THIS^.testConvertVolume(
	sourceValue := 1.0,
	sourceUnit := CNM_RecipeHandling.VolumeUnit.LITER,
	sourcePrefix := CNM_RecipeHandling.MetricPrefixes.NONE,
	expectedValue := 1000.0,
	expectedUnit := CNM_RecipeHandling.VolumeUnit.LITER,
	expectedPrefix:= CNM_RecipeHandling.MetricPrefixes.MILLI
);
THIS^.testConvertVolume(
	sourceValue := 1.0,
	sourceUnit := CNM_RecipeHandling.VolumeUnit.LITER,
	sourcePrefix := CNM_RecipeHandling.MetricPrefixes.NONE,
	expectedValue := 0.001,
	expectedUnit := CNM_RecipeHandling.VolumeUnit.CUBIC_METER,
	expectedPrefix:= CNM_RecipeHandling.MetricPrefixes.NONE
);
THIS^.testConvertVolume(
	sourceValue := 1.0,
	sourceUnit := CNM_RecipeHandling.VolumeUnit.LITER,
	sourcePrefix := CNM_RecipeHandling.MetricPrefixes.NONE,
	expectedValue := 0.264172 ,
	expectedUnit := CNM_RecipeHandling.VolumeUnit.US_GALLON,
	expectedPrefix:= CNM_RecipeHandling.MetricPrefixes.NONE
);
THIS^.testConvertVolume(
	sourceValue := 1.0,
	sourceUnit := CNM_RecipeHandling.VolumeUnit.LITER,
	sourcePrefix := CNM_RecipeHandling.MetricPrefixes.NONE,
	expectedValue := 0.219969 ,
	expectedUnit := CNM_RecipeHandling.VolumeUnit.US_DRY_GALLON,
	expectedPrefix:= CNM_RecipeHandling.MetricPrefixes.NONE
);
THIS^.testConvertVolume(
	sourceValue := 1.0,
	sourceUnit := CNM_RecipeHandling.VolumeUnit.LITER,
	sourcePrefix := CNM_RecipeHandling.MetricPrefixes.NONE,
	expectedValue := 1.8161708314990030466 ,
	expectedUnit := CNM_RecipeHandling.VolumeUnit.US_DRY_PINT,
	expectedPrefix:= CNM_RecipeHandling.MetricPrefixes.NONE
);
THIS^.testConvertVolume(
	sourceValue := 1.0,
	sourceUnit := CNM_RecipeHandling.VolumeUnit.US_DRY_PINT,
	sourcePrefix := CNM_RecipeHandling.MetricPrefixes.NONE,
	expectedValue :=  1.16365 ,
	expectedUnit := CNM_RecipeHandling.VolumeUnit.US_PINT,
	expectedPrefix:= CNM_RecipeHandling.MetricPrefixes.NONE
);
THIS^.testConvertVolume(
	sourceValue := 1.0,
	sourceUnit := CNM_RecipeHandling.VolumeUnit.LITER,
	sourcePrefix := CNM_RecipeHandling.MetricPrefixes.NONE,
	expectedValue :=  0.00130795,
	expectedUnit := CNM_RecipeHandling.VolumeUnit.US_CUBIC_YARD,
	expectedPrefix:= CNM_RecipeHandling.MetricPrefixes.NONE
);
THIS^.testConvertVolume(
	sourceValue := 1.0,
	sourceUnit := CNM_RecipeHandling.VolumeUnit.LITER,
	sourcePrefix := CNM_RecipeHandling.MetricPrefixes.NONE,
	expectedValue :=  0.03531467,
	expectedUnit := CNM_RecipeHandling.VolumeUnit.US_CUBIC_FOOT,
	expectedPrefix:= CNM_RecipeHandling.MetricPrefixes.NONE
);
THIS^.testConvertVolume(
	sourceValue := 0.0,
	sourceUnit := CNM_RecipeHandling.VolumeUnit.LITER,
	sourcePrefix := CNM_RecipeHandling.MetricPrefixes.NONE,
	expectedValue :=  0.0,
	expectedUnit := CNM_RecipeHandling.VolumeUnit.LITER,
	expectedPrefix:= CNM_RecipeHandling.MetricPrefixes.MILLI
);
THIS^.testConvertVolume(
	sourceValue := 0.0,
	sourceUnit := CNM_RecipeHandling.VolumeUnit.LITER,
	sourcePrefix := CNM_RecipeHandling.MetricPrefixes.NONE,
	expectedValue :=  0.0,
	expectedUnit := CNM_RecipeHandling.VolumeUnit.US_GALLON,
	expectedPrefix:= CNM_RecipeHandling.MetricPrefixes.MILLI
);
THIS^.testConvertVolume(
	sourceValue := 0.0,
	sourceUnit := CNM_RecipeHandling.VolumeUnit.LITER,
	sourcePrefix := CNM_RecipeHandling.MetricPrefixes.NONE,
	expectedValue :=  0.0,
	expectedUnit := CNM_RecipeHandling.VolumeUnit.US_DRY_GALLON,
	expectedPrefix:= CNM_RecipeHandling.MetricPrefixes.MILLI
);
THIS^.testConvertVolume(
	sourceValue := 1000.0,
	sourceUnit := CNM_RecipeHandling.VolumeUnit.LITER,
	sourcePrefix := CNM_RecipeHandling.MetricPrefixes.NONE,
	expectedValue :=  1000000.0,
	expectedUnit := CNM_RecipeHandling.VolumeUnit.LITER,
	expectedPrefix:= CNM_RecipeHandling.MetricPrefixes.MILLI
);
THIS^.testConvertVolume(
	sourceValue := 1000.0,
	sourceUnit := CNM_RecipeHandling.VolumeUnit.LITER,
	sourcePrefix := CNM_RecipeHandling.MetricPrefixes.NONE,
	expectedValue :=  1.0,
	expectedUnit := CNM_RecipeHandling.VolumeUnit.CUBIC_METER,
	expectedPrefix:= CNM_RecipeHandling.MetricPrefixes.NONE
);
THIS^.testConvertVolume(
	sourceValue := 1000.0,
	sourceUnit := CNM_RecipeHandling.VolumeUnit.LITER,
	sourcePrefix := CNM_RecipeHandling.MetricPrefixes.NONE,
	expectedValue := 264.172,
	expectedUnit := CNM_RecipeHandling.VolumeUnit.US_GALLON,
	expectedPrefix:= CNM_RecipeHandling.MetricPrefixes.NONE
);
THIS^.testConvertVolume(
	sourceValue := 1000.0,
	sourceUnit := CNM_RecipeHandling.VolumeUnit.LITER,
	sourcePrefix := CNM_RecipeHandling.MetricPrefixes.NONE,
	expectedValue := 227.020746,
	expectedUnit := CNM_RecipeHandling.VolumeUnit.US_DRY_GALLON,
	expectedPrefix:= CNM_RecipeHandling.MetricPrefixes.NONE
);
THIS^.testConvertVolume(
	sourceValue := -1.0,
	sourceUnit := CNM_RecipeHandling.VolumeUnit.LITER,
	sourcePrefix := CNM_RecipeHandling.MetricPrefixes.NONE,
	expectedValue := -1000.0,
	expectedUnit := CNM_RecipeHandling.VolumeUnit.LITER,
	expectedPrefix:= CNM_RecipeHandling.MetricPrefixes.MILLI
);
THIS^.testConvertVolume(
	sourceValue := -1.0,
	sourceUnit := CNM_RecipeHandling.VolumeUnit.LITER,
	sourcePrefix := CNM_RecipeHandling.MetricPrefixes.NONE,
	expectedValue := -0.264172,
	expectedUnit := CNM_RecipeHandling.VolumeUnit.US_GALLON,
	expectedPrefix:= CNM_RecipeHandling.MetricPrefixes.NONE
);
THIS^.testConvertVolume(
	sourceValue := 1.0,
	sourceUnit := CNM_RecipeHandling.VolumeUnit.LITER,
	sourcePrefix := CNM_RecipeHandling.MetricPrefixes.KILO,
	expectedValue := 0.26417205,
	expectedUnit := CNM_RecipeHandling.VolumeUnit.US_GALLON,
	expectedPrefix:= CNM_RecipeHandling.MetricPrefixes.KILO
);
THIS^.testConvertVolume(
	sourceValue := 1.0,
	sourceUnit := CNM_RecipeHandling.VolumeUnit.CUBIC_METER,
	sourcePrefix := CNM_RecipeHandling.MetricPrefixes.NONE,
	expectedValue := 6.28981,
	expectedUnit := CNM_RecipeHandling.VolumeUnit.US_OIL_BARREL,
	expectedPrefix:= CNM_RecipeHandling.MetricPrefixes.NONE
);
THIS^.testConvertVolume(
	sourceValue := 1.0,
	sourceUnit := CNM_RecipeHandling.VolumeUnit.CUBIC_METER,
	sourcePrefix := CNM_RecipeHandling.MetricPrefixes.KILO,
	expectedValue := 6289810771.5398332750,
	expectedUnit := CNM_RecipeHandling.VolumeUnit.US_OIL_BARREL,
	expectedPrefix:= CNM_RecipeHandling.MetricPrefixes.NONE
);
THIS^.testConvertVolume(
	sourceValue := 3.14,
	sourceUnit := CNM_RecipeHandling.VolumeUnit.CUBIC_METER,
	sourcePrefix := CNM_RecipeHandling.MetricPrefixes.NONE,
	expectedValue := 19.75,
	expectedUnit := CNM_RecipeHandling.VolumeUnit.US_OIL_BARREL,
	expectedPrefix:= CNM_RecipeHandling.MetricPrefixes.NONE
);
THIS^.testConvertVolume(
	sourceValue := 1.41,
	sourceUnit := CNM_RecipeHandling.VolumeUnit.LITER,
	sourcePrefix := CNM_RecipeHandling.MetricPrefixes.NONE,
	expectedValue := 0.0088937924,
	expectedUnit := CNM_RecipeHandling.VolumeUnit.US_OIL_BARREL,
	expectedPrefix:= CNM_RecipeHandling.MetricPrefixes.NONE
);
THIS^.testConvertVolume(
	sourceValue := 1.0,
	sourceUnit := CNM_RecipeHandling.VolumeUnit.US_OIL_BARREL,
	sourcePrefix := CNM_RecipeHandling.MetricPrefixes.NONE,
	expectedValue := 0.1589872949,
	expectedUnit := CNM_RecipeHandling.VolumeUnit.CUBIC_METER,
	expectedPrefix:= CNM_RecipeHandling.MetricPrefixes.NONE
);
THIS^.testConvertVolume(
	sourceValue := 3.14,
	sourceUnit := CNM_RecipeHandling.VolumeUnit.US_OIL_BARREL,
	sourcePrefix := CNM_RecipeHandling.MetricPrefixes.NONE,
	expectedValue := 16880.6289,
	expectedUnit := CNM_RecipeHandling.VolumeUnit.US_FLUID_OUNCE,
	expectedPrefix:= CNM_RecipeHandling.MetricPrefixes.NONE
);
THIS^.testConvertVolume(
	sourceValue := THIS^.MINUS_ZERO,
	sourceUnit := CNM_RecipeHandling.VolumeUnit.LITER,
	sourcePrefix := CNM_RecipeHandling.MetricPrefixes.KILO,
	expectedValue := THIS^.MINUS_ZERO,
	expectedUnit := CNM_RecipeHandling.VolumeUnit.US_GALLON,
	expectedPrefix:= CNM_RecipeHandling.MetricPrefixes.KILO
);
THIS^.testConvertVolume(
	sourceValue := THIS^.MIN_SUBNORMAL,
	sourceUnit := CNM_RecipeHandling.VolumeUnit.LITER,
	sourcePrefix := CNM_RecipeHandling.MetricPrefixes.KILO,
	expectedValue := THIS^.MIN_SUBNORMAL,
	expectedUnit := CNM_RecipeHandling.VolumeUnit.US_GALLON,
	expectedPrefix:= CNM_RecipeHandling.MetricPrefixes.KILO
);
THIS^.testConvertVolume(
	sourceValue := THIS^.MAX_SUBNORMAL,
	sourceUnit := CNM_RecipeHandling.VolumeUnit.LITER,
	sourcePrefix := CNM_RecipeHandling.MetricPrefixes.KILO,
	expectedValue := THIS^.MAX_SUBNORMAL,
	expectedUnit := CNM_RecipeHandling.VolumeUnit.US_GALLON,
	expectedPrefix:= CNM_RecipeHandling.MetricPrefixes.KILO
);
THIS^.testConvertVolume(
	sourceValue := THIS^.SMALLEST_NEGATIVE_SUBNORMAL,
	sourceUnit := CNM_RecipeHandling.VolumeUnit.LITER,
	sourcePrefix := CNM_RecipeHandling.MetricPrefixes.KILO,
	expectedValue := THIS^.SMALLEST_NEGATIVE_SUBNORMAL,
	expectedUnit := CNM_RecipeHandling.VolumeUnit.US_GALLON,
	expectedPrefix:= CNM_RecipeHandling.MetricPrefixes.KILO
);
THIS^.testConvertVolume(
	sourceValue := THIS^.SMALLEST_POSITIVE_SUBNORMAL,
	sourceUnit := CNM_RecipeHandling.VolumeUnit.LITER,
	sourcePrefix := CNM_RecipeHandling.MetricPrefixes.KILO,
	expectedValue := THIS^.SMALLEST_POSITIVE_SUBNORMAL,
	expectedUnit := CNM_RecipeHandling.VolumeUnit.US_GALLON,
	expectedPrefix:= CNM_RecipeHandling.MetricPrefixes.KILO
);
THIS^.testConvertVolumeSpecialCases(
	sourceValue := THIS^.NAN,
	sourceUnit := CNM_RecipeHandling.VolumeUnit.LITER,
	sourcePrefix := CNM_RecipeHandling.MetricPrefixes.KILO,
	expectedValue := THIS^.NAN,
	expectedUnit := CNM_RecipeHandling.VolumeUnit.US_GALLON,
	expectedPrefix:= CNM_RecipeHandling.MetricPrefixes.KILO
);
THIS^.testConvertVolumeSpecialCases(
	sourceValue := THIS^.INF,
	sourceUnit := CNM_RecipeHandling.VolumeUnit.LITER,
	sourcePrefix := CNM_RecipeHandling.MetricPrefixes.KILO,
	expectedValue := THIS^.INF,
	expectedUnit := CNM_RecipeHandling.VolumeUnit.US_GALLON,
	expectedPrefix:= CNM_RecipeHandling.MetricPrefixes.KILO
);
THIS^.testConvertVolumeSpecialCases(
	sourceValue := THIS^.MINUS_INF,
	sourceUnit := CNM_RecipeHandling.VolumeUnit.LITER,
	sourcePrefix := CNM_RecipeHandling.MetricPrefixes.KILO,
	expectedValue := THIS^.MINUS_INF,
	expectedUnit := CNM_RecipeHandling.VolumeUnit.US_GALLON,
	expectedPrefix:= CNM_RecipeHandling.MetricPrefixes.KILO
);
TcUnit.TEST_FINISHED();
END_METHOD

(*

short summary
==================
This test method tests ``ConvertWeight``
method of CNM_RecipeHandling library with various inputs

.. <legal notes>

legal notes
=================
| SPDX-FileCopyrightText: © 2025 ekvip automation GmbH <info@ekvip.de>
| SPDX-License-Identifier: Apache-2.0
| For details check: Apache-2.0_

.. _Apache-2.0: https://www.apache.org/licenses/LICENSE-2.0

.. </legal notes>

*)

METHOD runConvertWeight
VAR_INPUT
END_VAR
RETURN(NOT TcUnit.TEST_ORDERED('testConvertWeight'));

THIS^.testConvertWeight(
	sourceWeightValue := 1.0,
	sourceWeightUnit := CNM_RecipeHandling.WeightUnit.GRAM,
	sourcePrefix := CNM_RecipeHandling.MetricPrefixes.NONE,
	expectedValue := 1.0,
	expectedUnit := CNM_RecipeHandling.WeightUnit.GRAM,
	expectedPrefix:= CNM_RecipeHandling.MetricPrefixes.NONE
);
THIS^.testConvertWeight(
	sourceWeightValue := 1.0,
	sourceWeightUnit := CNM_RecipeHandling.WeightUnit.GRAM,
	sourcePrefix := CNM_RecipeHandling.MetricPrefixes.KILO,
	expectedValue := 1000.0,
	expectedUnit := CNM_RecipeHandling.WeightUnit.GRAM,
	expectedPrefix:= CNM_RecipeHandling.MetricPrefixes.NONE
);
THIS^.testConvertWeight(
	sourceWeightValue := 1.0,
	sourceWeightUnit := CNM_RecipeHandling.WeightUnit.GRAM,
	sourcePrefix := CNM_RecipeHandling.MetricPrefixes.KILO,
	expectedValue := 1000.0,
	expectedUnit := CNM_RecipeHandling.WeightUnit.GRAM,
	expectedPrefix:= CNM_RecipeHandling.MetricPrefixes.NONE
);
THIS^.testConvertWeight(
	sourceWeightValue := 1.0,
	sourceWeightUnit := CNM_RecipeHandling.WeightUnit.GRAM,
	sourcePrefix := CNM_RecipeHandling.MetricPrefixes.KILO,
	expectedValue := 0.001,
	expectedUnit := CNM_RecipeHandling.WeightUnit.TON,
	expectedPrefix:= CNM_RecipeHandling.MetricPrefixes.NONE
);
THIS^.testConvertWeight(
	sourceWeightValue := 0.001,
	sourceWeightUnit := CNM_RecipeHandling.WeightUnit.TON,
	sourcePrefix := CNM_RecipeHandling.MetricPrefixes.NONE,
	expectedValue := 2.20462,
	expectedUnit := CNM_RecipeHandling.WeightUnit.US_POUND,
	expectedPrefix:= CNM_RecipeHandling.MetricPrefixes.NONE
);
THIS^.testConvertWeight(
	sourceWeightValue := 1.0,
	sourceWeightUnit := CNM_RecipeHandling.WeightUnit.GRAM,
	sourcePrefix := CNM_RecipeHandling.MetricPrefixes.KILO,
	expectedValue := 35.274,
	expectedUnit := CNM_RecipeHandling.WeightUnit.US_OUNCE,
	expectedPrefix:= CNM_RecipeHandling.MetricPrefixes.NONE
);
THIS^.testConvertWeight(
	sourceWeightValue := 1.0,
	sourceWeightUnit := CNM_RecipeHandling.WeightUnit.GRAM,
	sourcePrefix := CNM_RecipeHandling.MetricPrefixes.NONE,
	expectedValue := 1000,
	expectedUnit := CNM_RecipeHandling.WeightUnit.GRAM,
	expectedPrefix:= CNM_RecipeHandling.MetricPrefixes.MILLI
);
THIS^.testConvertWeight(
	sourceWeightValue := 1.0,
	sourceWeightUnit := CNM_RecipeHandling.WeightUnit.GRAM,
	sourcePrefix := CNM_RecipeHandling.MetricPrefixes.NONE,
	expectedValue := 0.00220462,
	expectedUnit := CNM_RecipeHandling.WeightUnit.US_POUND,
	expectedPrefix:= CNM_RecipeHandling.MetricPrefixes.NONE
);
THIS^.testConvertWeight(
	sourceWeightValue := 1.0,
	sourceWeightUnit := CNM_RecipeHandling.WeightUnit.GRAM,
	sourcePrefix := CNM_RecipeHandling.MetricPrefixes.NONE,
	expectedValue := 0.035274,
	expectedUnit := CNM_RecipeHandling.WeightUnit.US_OUNCE,
	expectedPrefix:= CNM_RecipeHandling.MetricPrefixes.NONE
);
THIS^.testConvertWeight(
	sourceWeightValue := 0.0,
	sourceWeightUnit := CNM_RecipeHandling.WeightUnit.GRAM,
	sourcePrefix := CNM_RecipeHandling.MetricPrefixes.KILO,
	expectedValue := 0.0,
	expectedUnit := CNM_RecipeHandling.WeightUnit.GRAM,
	expectedPrefix:= CNM_RecipeHandling.MetricPrefixes.NONE
);
THIS^.testConvertWeight(
	sourceWeightValue := 0.0,
	sourceWeightUnit := CNM_RecipeHandling.WeightUnit.GRAM,
	sourcePrefix := CNM_RecipeHandling.MetricPrefixes.KILO,
	expectedValue := 0.0,
	expectedUnit := CNM_RecipeHandling.WeightUnit.US_POUND,
	expectedPrefix:= CNM_RecipeHandling.MetricPrefixes.NONE
);
THIS^.testConvertWeight(
	sourceWeightValue := 1000.0,
	sourceWeightUnit := CNM_RecipeHandling.WeightUnit.GRAM,
	sourcePrefix := CNM_RecipeHandling.MetricPrefixes.KILO,
	expectedValue := 1.0,
	expectedUnit := CNM_RecipeHandling.WeightUnit.TON,
	expectedPrefix:= CNM_RecipeHandling.MetricPrefixes.NONE
);
THIS^.testConvertWeight(
	sourceWeightValue := 1000.0,
	sourceWeightUnit := CNM_RecipeHandling.WeightUnit.GRAM,
	sourcePrefix := CNM_RecipeHandling.MetricPrefixes.KILO,
	expectedValue := 2204.62,
	expectedUnit := CNM_RecipeHandling.WeightUnit.US_POUND,
	expectedPrefix:= CNM_RecipeHandling.MetricPrefixes.NONE
);
THIS^.testConvertWeight(
	sourceWeightValue := 1000.0,
	sourceWeightUnit := CNM_RecipeHandling.WeightUnit.GRAM,
	sourcePrefix := CNM_RecipeHandling.MetricPrefixes.KILO,
	expectedValue := 35273.96195,
	expectedUnit := CNM_RecipeHandling.WeightUnit.US_OUNCE,
	expectedPrefix:= CNM_RecipeHandling.MetricPrefixes.NONE
);
THIS^.testConvertWeight(
	sourceWeightValue := -1.0,
	sourceWeightUnit := CNM_RecipeHandling.WeightUnit.GRAM,
	sourcePrefix := CNM_RecipeHandling.MetricPrefixes.KILO,
	expectedValue := -1000,
	expectedUnit := CNM_RecipeHandling.WeightUnit.GRAM,
	expectedPrefix:= CNM_RecipeHandling.MetricPrefixes.NONE
);
THIS^.testConvertWeight(
	sourceWeightValue := -1.0,
	sourceWeightUnit := CNM_RecipeHandling.WeightUnit.GRAM,
	sourcePrefix := CNM_RecipeHandling.MetricPrefixes.KILO,
	expectedValue := -35.274,
	expectedUnit := CNM_RecipeHandling.WeightUnit.US_OUNCE,
	expectedPrefix:= CNM_RecipeHandling.MetricPrefixes.NONE
);
THIS^.testConvertWeight(
	sourceWeightValue := 1.0,
	sourceWeightUnit := CNM_RecipeHandling.WeightUnit.GRAM,
	sourcePrefix := CNM_RecipeHandling.MetricPrefixes.MEGA,
	expectedValue := 1000.0,
	expectedUnit := CNM_RecipeHandling.WeightUnit.GRAM,
	expectedPrefix:= CNM_RecipeHandling.MetricPrefixes.KILO
);
THIS^.testConvertWeight(
	sourceWeightValue := 1.0,
	sourceWeightUnit := CNM_RecipeHandling.WeightUnit.GRAM,
	sourcePrefix := CNM_RecipeHandling.MetricPrefixes.HECTO,
	expectedValue := 100.0,
	expectedUnit := CNM_RecipeHandling.WeightUnit.GRAM,
	expectedPrefix:= CNM_RecipeHandling.MetricPrefixes.NONE
);
THIS^.testConvertWeight(
	sourceWeightValue := 1.0,
	sourceWeightUnit := CNM_RecipeHandling.WeightUnit.GRAM,
	sourcePrefix := CNM_RecipeHandling.MetricPrefixes.DEKA,
	expectedValue := 10.0,
	expectedUnit := CNM_RecipeHandling.WeightUnit.GRAM,
	expectedPrefix:= CNM_RecipeHandling.MetricPrefixes.NONE
);
THIS^.testConvertWeight(
	sourceWeightValue := 1.0,
	sourceWeightUnit := CNM_RecipeHandling.WeightUnit.GRAM,
	sourcePrefix := CNM_RecipeHandling.MetricPrefixes.DECI,
	expectedValue := 0.1,
	expectedUnit := CNM_RecipeHandling.WeightUnit.GRAM,
	expectedPrefix:= CNM_RecipeHandling.MetricPrefixes.NONE
);
THIS^.testConvertWeight(
	sourceWeightValue := 1.0,
	sourceWeightUnit := CNM_RecipeHandling.WeightUnit.GRAM,
	sourcePrefix := CNM_RecipeHandling.MetricPrefixes.CENTI,
	expectedValue := 0.01,
	expectedUnit := CNM_RecipeHandling.WeightUnit.GRAM,
	expectedPrefix:= CNM_RecipeHandling.MetricPrefixes.NONE
);
THIS^.testConvertWeight(
	sourceWeightValue := 1.0,
	sourceWeightUnit := CNM_RecipeHandling.WeightUnit.GRAM,
	sourcePrefix := CNM_RecipeHandling.MetricPrefixes.KILO,
	expectedValue := 0.03527396,
	expectedUnit := CNM_RecipeHandling.WeightUnit.US_OUNCE,
	expectedPrefix:= CNM_RecipeHandling.MetricPrefixes.KILO
);
THIS^.testConvertWeight(
	sourceWeightValue := THIS^.MINUS_ZERO,
	sourceWeightUnit := CNM_RecipeHandling.WeightUnit.GRAM,
	sourcePrefix := CNM_RecipeHandling.MetricPrefixes.KILO,
	expectedValue := THIS^.MINUS_ZERO,
	expectedUnit := CNM_RecipeHandling.WeightUnit.GRAM,
	expectedPrefix:= CNM_RecipeHandling.MetricPrefixes.MILLI
);
THIS^.testConvertWeight(
	sourceWeightValue := THIS^.MIN_SUBNORMAL,
	sourceWeightUnit := CNM_RecipeHandling.WeightUnit.GRAM,
	sourcePrefix := CNM_RecipeHandling.MetricPrefixes.KILO,
	expectedValue := THIS^.MIN_SUBNORMAL,
	expectedUnit := CNM_RecipeHandling.WeightUnit.GRAM,
	expectedPrefix:= CNM_RecipeHandling.MetricPrefixes.MILLI
);
THIS^.testConvertWeight(
	sourceWeightValue := THIS^.MAX_SUBNORMAL,
	sourceWeightUnit := CNM_RecipeHandling.WeightUnit.GRAM,
	sourcePrefix := CNM_RecipeHandling.MetricPrefixes.KILO,
	expectedValue := THIS^.MAX_SUBNORMAL,
	expectedUnit := CNM_RecipeHandling.WeightUnit.GRAM,
	expectedPrefix:= CNM_RecipeHandling.MetricPrefixes.MILLI
);
THIS^.testConvertWeight(
	sourceWeightValue := THIS^.SMALLEST_NEGATIVE_SUBNORMAL,
	sourceWeightUnit := CNM_RecipeHandling.WeightUnit.GRAM,
	sourcePrefix := CNM_RecipeHandling.MetricPrefixes.KILO,
	expectedValue := THIS^.SMALLEST_NEGATIVE_SUBNORMAL,
	expectedUnit := CNM_RecipeHandling.WeightUnit.GRAM,
	expectedPrefix:= CNM_RecipeHandling.MetricPrefixes.MILLI
);
THIS^.testConvertWeight(
	sourceWeightValue := THIS^.SMALLEST_POSITIVE_SUBNORMAL,
	sourceWeightUnit := CNM_RecipeHandling.WeightUnit.GRAM,
	sourcePrefix := CNM_RecipeHandling.MetricPrefixes.KILO,
	expectedValue := THIS^.SMALLEST_POSITIVE_SUBNORMAL,
	expectedUnit := CNM_RecipeHandling.WeightUnit.GRAM,
	expectedPrefix:= CNM_RecipeHandling.MetricPrefixes.MILLI
);
THIS^.testConvertWightSpecialCases(
	sourceWeightValue := THIS^.NAN,
	sourceWeightUnit := CNM_RecipeHandling.WeightUnit.GRAM,
	sourcePrefix := CNM_RecipeHandling.MetricPrefixes.KILO,
	expectedValue := THIS^.NAN,
	expectedUnit := CNM_RecipeHandling.WeightUnit.GRAM,
	expectedPrefix:= CNM_RecipeHandling.MetricPrefixes.MILLI
);
THIS^.testConvertWightSpecialCases(
	sourceWeightValue := THIS^.INF,
	sourceWeightUnit := CNM_RecipeHandling.WeightUnit.GRAM,
	sourcePrefix := CNM_RecipeHandling.MetricPrefixes.KILO,
	expectedValue := THIS^.INF,
	expectedUnit := CNM_RecipeHandling.WeightUnit.GRAM,
	expectedPrefix:= CNM_RecipeHandling.MetricPrefixes.MILLI
);
THIS^.testConvertWightSpecialCases(
	sourceWeightValue := THIS^.MINUS_INF,
	sourceWeightUnit := CNM_RecipeHandling.WeightUnit.GRAM,
	sourcePrefix := CNM_RecipeHandling.MetricPrefixes.KILO,
	expectedValue := THIS^.MINUS_INF,
	expectedUnit := CNM_RecipeHandling.WeightUnit.GRAM,
	expectedPrefix:= CNM_RecipeHandling.MetricPrefixes.MILLI
);
TcUnit.TEST_FINISHED();
END_METHOD

(*

short summary
==================
This test method tests ``FastPow10``
method of CNM_RecipeHandling library with various inputs

.. <legal notes>

legal notes
=================
| SPDX-FileCopyrightText: © 2025 ekvip automation GmbH <info@ekvip.de>
| SPDX-License-Identifier: Apache-2.0
| For details check: Apache-2.0_

.. _Apache-2.0: https://www.apache.org/licenses/LICENSE-2.0

.. </legal notes>

*)

METHOD runFastPow10
VAR_INPUT
END_VAR
RETURN(NOT TcUnit.TEST_ORDERED('testFastPow10'));
THIS^.testFastPow10(
	exponentValue := 32,
	expectedFastPow10Value := 100000000000000000000000000000000.0
);
THIS^.testFastPow10(
	exponentValue := -5,
	expectedFastPow10Value := 0.00001
);
THIS^.testFastPow10(
	exponentValue := -3,
	expectedFastPow10Value := 0.001
);
THIS^.testFastPow10(
	exponentValue := -1, 
	expectedFastPow10Value := 0.1
);
THIS^.testFastPow10(
	exponentValue := 0,
	expectedFastPow10Value := 1.0
);
THIS^.testFastPow10(
	exponentValue := 1,
	expectedFastPow10Value := 10.0
);
THIS^.testFastPow10(
	exponentValue := 2, 
	expectedFastPow10Value := 100.0
);
THIS^.testFastPow10(
	exponentValue := 3, 
	expectedFastPow10Value := 1000.0
);
THIS^.testFastPow10(
	exponentValue := 6, 
	expectedFastPow10Value := 1000000.0
);
THIS^.testFastPow10(
	exponentValue := 9, 
	expectedFastPow10Value := 1000000000.0
);
THIS^.testFastPow10(
	exponentValue := 12, 
	expectedFastPow10Value := 1000000000000.0
);
THIS^.testFastPow10(
	exponentValue := -6, 
	expectedFastPow10Value := 0.000001
);
THIS^.testFastPow10(
	exponentValue := -9, 
	expectedFastPow10Value := 0.000000001
);
THIS^.testFastPow10(
	exponentValue := -12,
	expectedFastPow10Value := 0.000000000001
);
THIS^.testFastPow10(
	exponentValue := 15, 
	expectedFastPow10Value := 1000000000000000.0
);
THIS^.testFastPow10(
	exponentValue := -15, 
	expectedFastPow10Value := 0.000000000000001
);
THIS^.testFastPow10(
	exponentValue := 0,
	expectedFastPow10Value := 1.0
);
TcUnit.TEST_FINISHED();
END_METHOD

(*

short summary
==================
This test method tests ``CalculateVelocity``
method of CNM_RecipeHandling library, 
it provides the possibility to handover test data via parameter 


.. <legal notes>

legal notes
=================
| SPDX-FileCopyrightText: © 2025 ekvip automation GmbH <info@ekvip.de>
| SPDX-License-Identifier: Apache-2.0
| For details check: Apache-2.0_

.. _Apache-2.0: https://www.apache.org/licenses/LICENSE-2.0

.. </legal notes>

parameters
==========

*)
METHOD testCalculateVelocity
VAR_INPUT
	(* The distance traveled, in raw value (e.g. 100.0) *)
	distanceDeltaValue : LREAL;
	(* The time it took to travel the distance (e.g. 10.0 seconds) *)
	timeDeltaValue : LREAL ;
	(* Unit of distance (e.g. METER, MILE) *)
	distanceUnit : CNM_RecipeHandling.LengthUnit;
	(* Unit of time (e.g. SECONDS, MINUTES) *)
	timeUnit: CNM_RecipeHandling.DurationUnit;
	(* Metric prefix for distance (e.g. KILO for kilometers) *)
	distancePrefix : CNM_RecipeHandling.MetricPrefixes;
	(* Metric prefix for time (e.g. MILLI for milliseconds) *)
	timePrefix : CNM_RecipeHandling.MetricPrefixes;
	(* Expected result of velocity calculation (e.g. 10.0) *)
	expectedVelocityValue : LREAL;
	(* Expected distance unit in result (e.g. METER) *)
	expectedDistanceUnit :CNM_RecipeHandling.LengthUnit;
	(* Expected metric prefix for distance (e.g. NONE) *)
	expectedDistancePrefix : CNM_RecipeHandling.MetricPrefixes;
	(* Expected time unit in result (e.g. SECONDS) *)
	expectedDurationUnit:CNM_RecipeHandling.DurationUnit;
	(*  Expected prefix for duration (e.g. MILLI) *)
	expectedDurationPrefix : CNM_RecipeHandling.MetricPrefixes;
	(* just the expectation if the assertion to test must be worng or true *)
	//assertionShouldBeTrue :BOOL;
END_VAR
VAR
	sourceDistance : CNM_RecipeHandling.Length;
	sourceTime : CNM_RecipeHandling.Duration;
	libResult : CNM_RecipeHandling.Velocity;
END_VAR

sourceTime.unit := timeUnit;
sourceTime.prefix := timePrefix; 

sourceDistance.value := distanceDeltaValue;
sourceDistance.unit := distanceUnit;
sourceDistance.prefix := distancePrefix;

sourceTime.value := timeDeltaValue;
sourceTime.unit := timeUnit;
sourceTime.prefix := timePrefix;


libResult := CNM_RecipeHandling.CalculateVelocity(
	distanceDelta :=sourceDistance,
	timeDelta := sourceTime,
);

THIS^.AssertEquals_LREAL(
    Expected := expectedVelocityValue,
    Actual := libResult.value,
    Delta := 0.01,
   Message := SEL(expectedVelocityValue = libResult.value,
	CONCAT('CalculateVelocity value fail: exp velocity = ',CONCAT( TO_STRING(expectedVelocityValue), concat( ', act velocity value = ', TO_STRING(libResult.value))))
    ,'test is ok'));

THIS^.AssertEquals_INT(
	Expected := expectedDistancePrefix,
	Actual := libResult.distancePrefix,
    Message := SEL(expectedDistancePrefix = libResult.distancePrefix,
	CONCAT('CalculateVelocity prefix fail: exp distance prefix  = ',CONCAT( TO_STRING(expectedDistancePrefix), concat( ', act distance prefix = ', TO_STRING(libResult.distancePrefix))))
    ,'test is ok')
);

THIS^.AssertEquals_INT(
	Expected := expectedDistanceUnit,
	Actual := libResult.distanceUnit,
    Message := SEL(expectedDistanceUnit = libResult.distanceUnit,
	CONCAT('CalculateVelocity unit fail: exp distance unit = ',CONCAT( TO_STRING(expectedDistanceUnit), concat( ', act distance unit = ', TO_STRING(libResult.distanceUnit))))
    ,'test is ok')
);

THIS^.AssertEquals_INT(
	Expected := expectedDurationPrefix,
	Actual := libResult.timePrefix,
    Message := SEL(expectedDurationPrefix = libResult.timePrefix,
	CONCAT('CalculateVelocity prefix fail: exp duration Prefix = ',CONCAT( TO_STRING(expectedDurationPrefix), concat( ', act duration Prefix = ', TO_STRING(libResult.timePrefix))))
    ,'test is ok')
);

THIS^.AssertEquals_INT(
	Expected := expectedDurationUnit,
	Actual := libResult.timeUnit,
    Message := SEL(expectedDurationUnit = libResult.timeUnit,
	CONCAT('CalculateVelocity unit fail: exp duration Unit = ',CONCAT( TO_STRING(expectedDurationUnit), concat( ', act duration Unit = ', TO_STRING(libResult.timeUnit))))
    ,'test is ok')
);
END_METHOD

(*

short summary
==================
This test method tests ``CalculateVelocity``
method of CNM_RecipeHandling library for special cases, 
it provides the possibility to handover test data via parameter 


.. <legal notes>

legal notes
=================
| SPDX-FileCopyrightText: © 2025 ekvip automation GmbH <info@ekvip.de>
| SPDX-License-Identifier: Apache-2.0
| For details check: Apache-2.0_

.. _Apache-2.0: https://www.apache.org/licenses/LICENSE-2.0

.. </legal notes>

parameters
==========

*)

METHOD testCalculateVelocitySpecialCases
	VAR_INPUT
	(* The distance traveled, in raw value (e.g. 100.0) *)
	distanceDeltaValue : LREAL;
	(* The time it took to travel the distance (e.g. 10.0 seconds) *)
	timeDeltaValue : LREAL ;
	(* Unit of distance (e.g. METER, MILE) *)
	distanceUnit : CNM_RecipeHandling.LengthUnit;
	(* Unit of time (e.g. SECONDS, MINUTES) *)
	timeUnit: CNM_RecipeHandling.DurationUnit;
	(* Metric prefix for distance (e.g. KILO for kilometers) *)
	distancePrefix : CNM_RecipeHandling.MetricPrefixes;
	(* Metric prefix for time (e.g. MILLI for milliseconds) *)
	timePrefix : CNM_RecipeHandling.MetricPrefixes;
	(* Expected result of velocity calculation (e.g. 10.0) *)
	expectedVelocityValue : LREAL;
	(* Expected distance unit in result (e.g. METER) *)
	expectedDistanceUnit :CNM_RecipeHandling.LengthUnit;
	(* Expected metric prefix for distance (e.g. NONE) *)
	expectedDistancePrefix : CNM_RecipeHandling.MetricPrefixes;
	(* Expected time unit in result (e.g. SECONDS) *)
	expectedDurationUnit:CNM_RecipeHandling.DurationUnit;
	(*  Expected prefix for duration (e.g. MILLI) *)
	expectedDurationPrefix : CNM_RecipeHandling.MetricPrefixes;;
END_VAR
VAR
	sourceDistance : CNM_RecipeHandling.Length;
	sourceTime : CNM_RecipeHandling.Duration;
	libResult : CNM_RecipeHandling.Velocity;
	(* contains the format string for the test message *)
	//message :Tc2_System.T_MaxString := 'Test failed';
	//Actual: INT;
END_VAR
sourceTime.unit := timeUnit;
sourceTime.prefix := timePrefix; 

sourceDistance.value := distanceDeltaValue;
sourceDistance.unit := distanceUnit;
sourceDistance.prefix := distancePrefix;

sourceTime.value := timeDeltaValue;
sourceTime.unit := timeUnit;
sourceTime.prefix := timePrefix;

libResult := CNM_RecipeHandling.CalculateVelocity(
	distanceDelta :=sourceDistance,
	timeDelta := sourceTime,
);

IF Tc2_Utilities.LrealIsNaN(expectedVelocityValue) THEN
	AssertTrue(Condition := Tc2_Utilities.LrealIsNaN(libResult.value),
    Message := 'test faild assertion NaN should be true');
ELSIF NOT (Tc2_Utilities.LrealIsFinite(expectedVelocityValue))THEN
	 AssertTrue(Condition := NOT(Tc2_Utilities.LrealIsFinite(libResult.value)),
    Message := 'test faild assertion INF should be True');
END_IF
END_METHOD

METHOD testConvertAngle
VAR_INPUT
	(* The input value to convert (e.g. 3.14159) *)
	sourceValue : LREAL;
	(* The unit of the input angle (e.g. RADIANS, DEGREES) *)
	sourceUnit : CNM_RecipeHandling.AngleUnit;
	(* The expected result after conversion *)
	expectedValue : LREAL;
	(* The expected output unit *)
	expectedUnit :CNM_RecipeHandling.AngleUnit;
END_VAR
VAR
	sourceAngle : CNM_RecipeHandling.Angle;
	libResult : CNM_RecipeHandling.Angle;
	delta : LREAL;
END_VAR
// Setup test input
sourceAngle.value := sourceValue;
sourceAngle.unit := sourceUnit;

// Call the function to test
libResult := CNM_RecipeHandling.ConvertAngle(
	angleToConvert := sourceAngle,
	convertTo := expectedUnit
);

// Calculate appropriate delta based on magnitude of expected value
IF ABS(expectedValue) > 1000.0 THEN
	delta := 0.1; // Larger tolerance for large numbers (arc seconds)
ELSIF ABS(expectedValue) > 100.0 THEN
	delta := 0.01; // Medium tolerance for medium numbers
ELSIF ABS(expectedValue) > 1.0 THEN
	delta := 0.0001; // Small tolerance for normal numbers
ELSE
	delta := 0.000001; // Very small tolerance for small numbers
END_IF

// Verify the unit is correct
THIS^.AssertEquals_INT(
	Expected := expectedUnit,
	Actual := libResult.unit,
	Message := CONCAT('Unit conversion failed: expected ', 
		CONCAT(TO_STRING(expectedUnit), 
		CONCAT(', got ', TO_STRING(libResult.unit))))
);

// Verify the value is correct
THIS^.AssertEquals_LREAL(
	Expected := expectedValue,
	Actual := libResult.value,
	Delta := delta,
	Message := CONCAT('Value conversion failed: from ', 
		CONCAT(TO_STRING(sourceUnit), 
		CONCAT(', to ', TO_STRING(expectedUnit))))
);
END_METHOD

METHOD testConvertAngleSpecialCases
VAR_INPUT
	(* The input value to convert (e.g. NaN, Inf) *)
	sourceValue : LREAL;
	(* The unit of the input angle *)
	sourceUnit : CNM_RecipeHandling.AngleUnit;
	(* The expected result after conversion *)
	expectedValue : LREAL;
	(* The expected output unit *)
	expectedUnit :CNM_RecipeHandling.AngleUnit;
END_VAR
VAR
	sourceAngle : CNM_RecipeHandling.Angle;
	libResult : CNM_RecipeHandling.Angle;
END_VAR
// Setup test input
sourceAngle.value := sourceValue;
sourceAngle.unit := sourceUnit;

// Call the function to test
libResult := CNM_RecipeHandling.ConvertAngle(
	angleToConvert := sourceAngle,
	convertTo := expectedUnit
);

IF Tc2_Utilities.LrealIsNaN(expectedValue) THEN
	AssertTrue(Condition := Tc2_Utilities.LrealIsNaN(libResult.value),
    Message := 'test failed assertion NaN should be true');
ELSIF NOT (Tc2_Utilities.LrealIsFinite(expectedValue))THEN
	 AssertTrue(Condition := NOT(Tc2_Utilities.LrealIsFinite(libResult.value)),
    Message := 'test faild assertion INF should be True');
END_IF
END_METHOD

(*

short summary
==================
This test method tests ``ConvertAngularVelocity``
method of CNM_RecipeHandling library, 
it provides the possibility to handover test data via parameter 


.. <legal notes>

legal notes
=================
| SPDX-FileCopyrightText: © 2025 ekvip automation GmbH <info@ekvip.de>
| SPDX-License-Identifier: Apache-2.0
| For details check: Apache-2.0_

.. _Apache-2.0: https://www.apache.org/licenses/LICENSE-2.0

.. </legal notes>

parameters
==========

*)

METHOD testConvertAngularVelocity
VAR_INPUT
    (* Input velocity value to be converted, e.g. 10.0 *)
    sourceVelocityValue : LREAL; 
    (* Expected result after conversion, used for assertion *)
    expectedVelocityValue : LREAL;
    (* Unit of distance used in velocity, e.g. METER *)
    sourceUnit : CNM_RecipeHandling.AngleUnit;
    (* Expected unit of distance after conversion *)
    expectedAngleUnit : CNM_RecipeHandling.AngleUnit;
    (* Unit of time used in velocity, e.g. SECONDS *)
    sourceDurationUnit : CNM_RecipeHandling.DurationUnit;
    (* Metric prefix of the time input, e.g. MILLI *)
    sourceDurationPrefix : CNM_RecipeHandling.MetricPrefixes;
    (* Expected time unit after conversion *)
    expectedDurationUnit : CNM_RecipeHandling.DurationUnit;
    (* Expected time prefix after conversion *)
    expectedDurationPrefix : CNM_RecipeHandling.MetricPrefixes;
END_VAR
VAR
	sourceVelocity : CNM_RecipeHandling.AngularVelocity;
	libResult : CNM_RecipeHandling.AngularVelocity;
	sourcePrefix: CNM_RecipeHandling.MetricPrefixes;
END_VAR

//test-input
sourceVelocity.value := sourceVelocityValue;
sourceVelocity.angularDistanceUnit := sourceUnit;
sourceVelocity.timeUnit := sourceDurationUnit;
sourceVelocity.timePrefix := sourceDurationPrefix; 

//function to call
libResult := CNM_RecipeHandling.ConvertAngularVelocity(
	angularVelocityToConvert := sourceVelocity,
	convertAngleTo := expectedAngleUnit,
	convertTimeTo := expectedDurationUnit,
	resultPrefixTime := expectedDurationPrefix
);

THIS^.AssertEquals_LREAL(
    Expected := expectedVelocityValue,
    Actual := libResult.value,
    Delta := 0.01,
   Message := SEL(expectedVelocityValue = libResult.value,
	CONCAT('value fail: exp velocity value = ',CONCAT( TO_STRING(expectedVelocityValue), concat( ', act  velocity value = ', TO_STRING(libResult.value))))
    ,'test is ok'));

THIS^.AssertEquals_INT(
	Expected := expectedAngleUnit,
	Actual := libResult.angularDistanceUnit,
    Message := CONCAT('ConvertVelocity unit fail: exp distance unit = ',CONCAT( TO_STRING(expectedAngleUnit), concat( ', act distance unit = ', TO_STRING(libResult.angularDistanceUnit))))
);

THIS^.AssertEquals_INT(
	Expected := expectedDurationPrefix,
	Actual := libResult.timePrefix,
    Message := SEL(expectedDurationPrefix = libResult.timePrefix,
	CONCAT('ConvertVelocity prefix fail: exp duration Prefix = ',CONCAT( TO_STRING(expectedDurationPrefix), concat( ', act duration Prefix = ', TO_STRING(libResult.timePrefix))))
    ,'test is ok')
);
THIS^.AssertEquals_INT(
	Expected := expectedDurationUnit,
	Actual := libResult.timeUnit,
    Message := SEL(expectedDurationUnit = libResult.timeUnit,
	CONCAT('ConvertVelocity unit fail: exp duration Unit = ',CONCAT( TO_STRING(expectedDurationUnit), concat( ', act duration Unit = ', TO_STRING(libResult.timeUnit))))
    ,'test is ok')
);
END_METHOD

(*

short summary
==================
This test method tests ``ConvertVelocity``
method of CNM_RecipeHandling library for special cases, 
it provides the possibility to handover test data via parameter 


.. <legal notes>

legal notes
=================
| SPDX-FileCopyrightText: © 2025 ekvip automation GmbH <info@ekvip.de>
| SPDX-License-Identifier: Apache-2.0
| For details check: Apache-2.0_

.. _Apache-2.0: https://www.apache.org/licenses/LICENSE-2.0

.. </legal notes>

parameters
==========

*)

METHOD testConvertAngularVelocitySpecialCases
VAR_INPUT
    (* Input velocity value to be converted, e.g. 10.0 *)
    sourceVelocityValue : LREAL; 
    (* Expected result after conversion, used for assertion *)
    expectedVelocityValue : LREAL;
    (* Unit of distance used in velocity, e.g. METER *)
    sourceUnit : CNM_RecipeHandling.AngleUnit;
    (* Expected unit of distance after conversion *)
    expectedAngleUnit : CNM_RecipeHandling.AngleUnit;
    (* Unit of time used in velocity, e.g. SECONDS *)
    sourceDurationUnit : CNM_RecipeHandling.DurationUnit;
    (* Metric prefix of the time input, e.g. MILLI *)
    sourceDurationPrefix : CNM_RecipeHandling.MetricPrefixes;
    (* Expected time unit after conversion *)
    expectedDurationUnit : CNM_RecipeHandling.DurationUnit;
    (* Expected time prefix after conversion *)
    expectedDurationPrefix : CNM_RecipeHandling.MetricPrefixes;
END_VAR
VAR
	sourceVelocity : CNM_RecipeHandling.AngularVelocity;
	libResult : CNM_RecipeHandling.AngularVelocity;
	sourcePrefix: CNM_RecipeHandling.MetricPrefixes;
END_VAR
//test-input
sourceVelocity.value := sourceVelocityValue;
sourceVelocity.angularDistanceUnit := sourceUnit;
sourceVelocity.timeUnit := sourceDurationUnit;
sourceVelocity.timePrefix := sourceDurationPrefix; 

//function to call
libResult := CNM_RecipeHandling.ConvertAngularVelocity(
	angularVelocityToConvert:=sourceVelocity,
	convertAngleTo :=expectedAngleUnit,
	convertTimeTo := expectedDurationUnit,
	resultPrefixTime := expectedDurationPrefix
);

IF Tc2_Utilities.LrealIsNaN(expectedVelocityValue) THEN
	AssertTrue(Condition := Tc2_Utilities.LrealIsNaN(libResult.value),
    Message := 'test faild assertion NaN should be true');
ELSIF NOT (Tc2_Utilities.LrealIsFinite(expectedVelocityValue))THEN
	 AssertFalse(Condition := Tc2_Utilities.LrealIsFinite(libResult.value),
    Message := 'test faild assertion INF should be True');
END_IF
END_METHOD

(*

short summary
==================
This test method tests ``ConvertArea``
method of CNM_RecipeHandling library, 
it provides the possibility to handover test data via parameter 


.. <legal notes>

legal notes
=================
| SPDX-FileCopyrightText: © 2025 ekvip automation GmbH <info@ekvip.de>
| SPDX-License-Identifier: Apache-2.0
| For details check: Apache-2.0_

.. _Apache-2.0: https://www.apache.org/licenses/LICENSE-2.0

.. </legal notes>

parameters
==========

*)

METHOD testConvertArea
VAR_INPUT
	(* Input area value to be converted (e.g., 1.0) *)
	sourceValue : LREAL;
	(* Unit of the source area (e.g., SQUARE_METER, US_ACRE) *)
	sourceUnit : CNM_RecipeHandling.AreaUnit;
	(* Metric prefix of the source area unit (e.g., NONE, KILO, MILLI) *)
	sourcePrefix : CNM_RecipeHandling.MetricPrefixes;
	(* Expected result value after conversion *)
	expectedValue : LREAL;
	(* Target unit to which the area should be converted *)
	expectedUnit :CNM_RecipeHandling.AreaUnit;
	(* Metric prefix for the expected unit (e.g., NONE, MILLI) *)
	expectedPrefix : CNM_RecipeHandling.MetricPrefixes;
END_VAR
VAR
	sourceArea : CNM_RecipeHandling.Area;
	libResult : CNM_RecipeHandling.Area;
END_VAR
sourceArea.value := sourceValue;
sourceArea.unit := sourceUnit;
sourceArea.prefix := sourcePrefix;

libResult := CNM_RecipeHandling.ConvertArea(
	areaToconvert := sourceArea,
	convertTo := expectedUnit,
	resultPrefix := expectedPrefix
);

THIS^.AssertEquals_LREAL(
	Expected := expectedValue,
	Actual := libResult.value,
	Delta := 0.01,
   Message := SEL(expectedValue = libResult.value,
	CONCAT('normal case testConvertArea value fail: exp = ',CONCAT( TO_STRING(expectedValue), concat( ', act = ', TO_STRING(libResult.value))))
    ,'test is ok'))
;
THIS^.AssertEquals_INT(
	Expected := expectedPrefix,
	Actual := libResult.prefix,
    Message := SEL(expectedPrefix = libResult.prefix,
	CONCAT('normal case testConvertAre prefix fail: exp = ',CONCAT( TO_STRING(expectedPrefix), concat( ', act = ', TO_STRING(libResult.prefix))))
    ,'test is ok')
);

THIS^.AssertEquals_INT(
	Expected := expectedUnit,
	Actual := libResult.unit,
    Message := SEL(expectedUnit = libResult.unit,
	CONCAT('normal case testConvertAre unit fail: exp = ',CONCAT( TO_STRING(expectedUnit), concat( ', act = ', TO_STRING(libResult.unit))))
    ,'test is ok')
);
END_METHOD

(*

short summary
==================
This test method tests ``ConvertArea``
method of CNM_RecipeHandling library, 
it provides the possibility to handover test data via parameter 


.. <legal notes>

legal notes
=================
| SPDX-FileCopyrightText: © 2025 ekvip automation GmbH <info@ekvip.de>
| SPDX-License-Identifier: Apache-2.0
| For details check: Apache-2.0_

.. _Apache-2.0: https://www.apache.org/licenses/LICENSE-2.0

.. </legal notes>

parameters
==========

*)
METHOD testConvertAreaSpecialCases
VAR_INPUT
	(* Input area value to be converted (e.g., 1.0) *)
	sourceValue : LREAL;
	(* Unit of the source area (e.g., SQUARE_METER, US_ACRE) *)
	sourceUnit : CNM_RecipeHandling.AreaUnit;
	(* Metric prefix of the source area unit (e.g., NONE, KILO, MILLI) *)
	sourcePrefix : CNM_RecipeHandling.MetricPrefixes;
	(* Expected result value after conversion *)
	expectedValue : LREAL;
	(* Target unit to which the area should be converted *)
	expectedUnit :CNM_RecipeHandling.AreaUnit;
	(* Metric prefix for the expected unit (e.g., NONE, MILLI) *)
	expectedPrefix : CNM_RecipeHandling.MetricPrefixes;
END_VAR
VAR
	a :BOOL;
	input : CNM_RecipeHandling.Area;
	libResult : CNM_RecipeHandling.Area;
END_VAR
input.value := sourceValue;
input.unit := sourceUnit;
input.prefix := sourcePrefix;

libResult := CNM_RecipeHandling.ConvertArea(
	areaToconvert := input,
	convertTo := expectedUnit,
	resultPrefix := expectedPrefix
);

IF Tc2_Utilities.LrealIsNaN(expectedValue) THEN
	AssertTrue(Condition := Tc2_Utilities.LrealIsNaN(libResult.value),
    Message := 'test faild assertion NaN should be true');
ELSIF NOT (Tc2_Utilities.LrealIsFinite(expectedValue))THEN
	 AssertTrue(Condition := NOT(Tc2_Utilities.LrealIsFinite(libResult.value)),
    Message := 'test faild assertion INF should be True');
END_IF
END_METHOD

(*

short summary
==================
This test method tests ``ConvertDuration``
method of CNM_RecipeHandling library, 
it provides the possibility to handover test data via parameter 


.. <legal notes>

legal notes
=================
| SPDX-FileCopyrightText: © 2025 ekvip automation GmbH <info@ekvip.de>
| SPDX-License-Identifier: Apache-2.0
| For details check: Apache-2.0_

.. _Apache-2.0: https://www.apache.org/licenses/LICENSE-2.0

.. </legal notes>

parameters
==========

*)

METHOD testConvertDuration
VAR_INPUT
	(* The original time value to convert (e.g. 120.0) *)
	sourceValue : LREAL;
	(* The unit of the input time (e.g. SECONDS, MINUTES) *)
	sourceUnit : CNM_RecipeHandling.DurationUnit;
	(* The metric prefix for input time (e.g. MILLI for milliseconds) *)
	sourcePrefix : CNM_RecipeHandling.MetricPrefixes;
	(* The expected result value after conversion (e.g. 2.0) *)
	expectedValue : LREAL;
	(* The expected time unit after conversion (e.g. MINUTES) *)
	expectedUnit :CNM_RecipeHandling.DurationUnit;
	(* The expected metric prefix for the result (e.g. NONE) *)
	expectedPrefix : CNM_RecipeHandling.MetricPrefixes;
END_VAR
VAR
	sourceDuration : CNM_RecipeHandling.Duration;
	libResult : CNM_RecipeHandling.Duration;
END_VAR
sourceDuration.value := sourceValue;
sourceDuration.unit := sourceUnit;
sourceDuration.prefix := sourcePrefix;

libResult := CNM_RecipeHandling.ConvertDuration(
	durationToConvert :=sourceDuration,
	convertTo := expectedUnit,
	resultPrefix := expectedPrefix
);

THIS^.AssertEquals_LREAL(
    Expected := expectedValue,
    Actual := libResult.value,
    Delta := 0.01,
   Message := SEL(expectedValue = libResult.value,
	CONCAT('ConvertDuration value fail: exp = ',CONCAT( TO_STRING(expectedValue), concat( ', act = ', TO_STRING(libResult.value))))
    ,'test is ok'));

THIS^.AssertEquals_INT(
	Expected := expectedPrefix,
	Actual := libResult.prefix,
    Message := SEL(expectedPrefix = libResult.prefix,
	CONCAT('ConvertDuration prefix fail: exp = ',CONCAT( TO_STRING(expectedPrefix), concat( ', act = ', TO_STRING(libResult.prefix))))
    ,'test is ok')
);

THIS^.AssertEquals_INT(
	Expected := expectedUnit,
	Actual := libResult.unit,
    Message := SEL(expectedUnit = libResult.unit,
	CONCAT('ConvertDuration unit fail: exp = ',CONCAT( TO_STRING(expectedUnit), concat( ', act = ', TO_STRING(libResult.unit))))
    ,'test is ok')
);
END_METHOD

(*

short summary
==================
This test method tests ``ConvertDuration``
method of CNM_RecipeHandling library for special cases, 
it provides the possibility to handover test data via parameter 


.. <legal notes>

legal notes
=================
| SPDX-FileCopyrightText: © 2025 ekvip automation GmbH <info@ekvip.de>
| SPDX-License-Identifier: Apache-2.0
| For details check: Apache-2.0_

.. _Apache-2.0: https://www.apache.org/licenses/LICENSE-2.0

.. </legal notes>

parameters
==========

*)

METHOD testConvertDurationSpecialCases
VAR_INPUT
	(* The original time value to convert (e.g. 120.0) *)
	sourceValue : LREAL;
	(* The unit of the input time (e.g. SECONDS, MINUTES) *)
	sourceUnit : CNM_RecipeHandling.DurationUnit;
	(* The metric prefix for input time (e.g. MILLI for milliseconds) *)
	sourcePrefix : CNM_RecipeHandling.MetricPrefixes;
	(* The expected result value after conversion (e.g. 2.0) *)
	expectedValue : LREAL;
	(* The expected time unit after conversion (e.g. MINUTES) *)
	expectedUnit :CNM_RecipeHandling.DurationUnit;
	(* The expected metric prefix for the result (e.g. NONE) *)
	expectedPrefix : CNM_RecipeHandling.MetricPrefixes;
END_VAR
VAR
	sourceDuration : CNM_RecipeHandling.Duration;
	libResult : CNM_RecipeHandling.Duration;
END_VAR
sourceDuration.value := sourceValue;
sourceDuration.unit := sourceUnit;
sourceDuration.prefix := sourcePrefix;

libResult := CNM_RecipeHandling.ConvertDuration(
	durationToConvert :=sourceDuration,
	convertTo := expectedUnit,
	resultPrefix := expectedPrefix
);

IF Tc2_Utilities.LrealIsNaN(expectedValue) THEN
	AssertTrue(Condition := Tc2_Utilities.LrealIsNaN(libResult.value),
    Message := 'test faild assertion NaN should be true');
ELSIF NOT (Tc2_Utilities.LrealIsFinite(expectedValue))THEN
	 AssertTrue(Condition := NOT(Tc2_Utilities.LrealIsFinite(libResult.value)),
    Message := 'test faild assertion INF should be True');
END_IF
END_METHOD

(*

short summary
==================
This test method tests ``ConvertLength``
method of CNM_RecipeHandling library, 
it provides the possibility to handover test data via parameter 


.. <legal notes>

legal notes
=================
| SPDX-FileCopyrightText: © 2025 ekvip automation GmbH <info@ekvip.de>
| SPDX-License-Identifier: Apache-2.0
| For details check: Apache-2.0_

.. _Apache-2.0: https://www.apache.org/licenses/LICENSE-2.0

.. </legal notes>

parameters
==========

*)

METHOD testConvertLength
VAR_INPUT
	(* The input value to convert (e.g. 1.0) *)
	sourceValue : LREAL;
	(* The unit of the input length (e.g. METER, INCH) *)
	sourceUnit : CNM_RecipeHandling.LengthUnit;
	(* Metric prefix for the input value (e.g. MILLI, KILO) *)
	sourcePrefix : CNM_RecipeHandling.MetricPrefixes;
	(* The expected result after conversion (e.g. 1000.0) *)
	expectedValue : LREAL;
	(* The expected output unit (e.g. MILLIMETER) *)
	expectedUnit :CNM_RecipeHandling.LengthUnit;
	(* The expected metric prefix for the output (e.g. NONE) *)
	expectedPrefix : CNM_RecipeHandling.MetricPrefixes;
END_VAR
VAR
	sourceDistance : CNM_RecipeHandling.Length;
	libResult : CNM_RecipeHandling.Length;
END_VAR

//teat-input
sourceDistance.value := sourceValue;
sourceDistance.unit := sourceUnit;
sourceDistance.prefix := sourcePrefix;

//function to call
libResult := CNM_RecipeHandling.ConvertLength(
	lengthToConvert :=sourceDistance,
	convertTo := expectedUnit,
	resultPrefix := expectedPrefix
);

THIS^.AssertEquals_LREAL(
    Expected := expectedValue,
    Actual := libResult.value,
    Delta := 0.01,
   Message := SEL(expectedValue = libResult.value,
	CONCAT('ConvertLength value fail: exp = ',CONCAT( TO_STRING(expectedValue), concat( ', act = ', TO_STRING(libResult.value))))
    ,'test is ok'));


THIS^.AssertEquals_INT(
	Expected := expectedPrefix,
	Actual := libResult.prefix,
    Message := SEL(expectedPrefix = libResult.prefix,
	CONCAT('ConvertLength prefix fail: exp = ',CONCAT( TO_STRING(expectedPrefix), concat( ', act = ', TO_STRING(libResult.prefix))))
    ,'test is ok')
);
THIS^.AssertEquals_INT(
	Expected := expectedUnit,
	Actual := libResult.unit,
    Message := SEL(expectedUnit = libResult.unit,
	CONCAT('ConvertLength unit fail: exp = ',CONCAT( TO_STRING(expectedUnit), concat( ', act = ', TO_STRING(libResult.unit))))
    ,'test is ok')
);
END_METHOD

(*

short summary
==================
This test method tests ``ConvertLength``
method of CNM_RecipeHandling library for special cases, 
it provides the possibility to handover test data via parameter 


.. <legal notes>

legal notes
=================
| SPDX-FileCopyrightText: © 2025 ekvip automation GmbH <info@ekvip.de>
| SPDX-License-Identifier: Apache-2.0
| For details check: Apache-2.0_

.. _Apache-2.0: https://www.apache.org/licenses/LICENSE-2.0

.. </legal notes>

parameters
==========

*)
METHOD testConvertLengthSpecialCases
VAR_INPUT
	(* The input value to convert (e.g. 1.0) *)
	sourceValue : LREAL;
	(* The unit of the input length (e.g. METER, INCH) *)
	sourceUnit : CNM_RecipeHandling.LengthUnit;
	(* Metric prefix for the input value (e.g. MILLI, KILO) *)
	sourcePrefix : CNM_RecipeHandling.MetricPrefixes;
	(* The expected result after conversion (e.g. 1000.0) *)
	expectedValue : LREAL;
	(* The expected output unit (e.g. MILLIMETER) *)
	expectedUnit :CNM_RecipeHandling.LengthUnit;
	(* The expected metric prefix for the output (e.g. NONE) *)
	expectedPrefix : CNM_RecipeHandling.MetricPrefixes;
END_VAR
VAR
	sourceDistance : CNM_RecipeHandling.Length;
	libResult : CNM_RecipeHandling.Length;
END_VAR

//teat-input
sourceDistance.value := sourceValue;
sourceDistance.unit := sourceUnit;
sourceDistance.prefix := sourcePrefix;

//function to call
libResult := CNM_RecipeHandling.ConvertLength(
	lengthToConvert :=sourceDistance,
	convertTo := expectedUnit,
	resultPrefix := expectedPrefix
);

IF Tc2_Utilities.LrealIsNaN(expectedValue) THEN
	AssertTrue(Condition := Tc2_Utilities.LrealIsNaN(libResult.value),
    Message := 'test faild assertion NaN should be true');
ELSIF NOT (Tc2_Utilities.LrealIsFinite(expectedValue))THEN
	 AssertTrue(Condition := NOT(Tc2_Utilities.LrealIsFinite(libResult.value)),
    Message := 'test faild assertion INF should be True');
END_IF
END_METHOD

(*

short summary
==================
This test method tests ``ConvertPressure``
method of CNM_RecipeHandling library, 
it provides the possibility to handover test data via parameter 


.. <legal notes>

legal notes
=================
| SPDX-FileCopyrightText: © 2025 ekvip automation GmbH <info@ekvip.de>
| SPDX-License-Identifier: Apache-2.0
| For details check: Apache-2.0_

.. _Apache-2.0: https://www.apache.org/licenses/LICENSE-2.0

.. </legal notes>

parameters
==========

*)

METHOD testConvertPressure
VAR_INPUT
	(* The numeric pressure value to convert (e.g. 101325.0) *)
	sourceValue : LREAL;
	(* The original pressure unit (e.g. PASCAL, BAR) *)
	sourceUnit : CNM_RecipeHandling.PressureUnit;
	(*  Metric prefix for the input value (e.g. KILO, MILLI) *)
	sourcePrefix : CNM_RecipeHandling.MetricPrefixes;
	(* The expected result after conversion (e.g. 1.01325) *)
	expectedValue : LREAL;
	(* The target unit to which the pressure should be converted (e.g. BAR) *)
	expectedUnit :CNM_RecipeHandling.PressureUnit;
	(* Metric prefix for the expected result (e.g. NONE) *)
	expectedPrefix : CNM_RecipeHandling.MetricPrefixes;
END_VAR
VAR
	sourcePressure : CNM_RecipeHandling.Pressure;
	libResult : CNM_RecipeHandling.Pressure;
END_VAR

//test-input
sourcePressure.value := sourceValue;
sourcePressure.unit := sourceUnit;
sourcePressure.prefix := sourcePrefix;

//function to call
libResult := CNM_RecipeHandling.ConvertPressure(
	pressureToConvert :=sourcePressure,
	convertTo := expectedUnit,
	resultPrefix := expectedPrefix
);

THIS^.AssertEquals_LREAL(
    Expected := expectedValue,
    Actual := libResult.value,
    Delta := 0.01,
   Message := SEL(expectedValue = libResult.value,
	CONCAT('Pressure value fail: exp = ',CONCAT( TO_STRING(expectedValue), concat( ', act = ', TO_STRING(libResult.value))))
    ,'test is ok'));


THIS^.AssertEquals_INT(
	Expected := expectedPrefix,
	Actual := libResult.prefix,
    Message := SEL(expectedPrefix = libResult.prefix,
	CONCAT('Pressure prefix fail: exp = ',CONCAT( TO_STRING(expectedPrefix), concat( ', act = ', TO_STRING(libResult.prefix))))
    ,'test is ok')
);
THIS^.AssertEquals_INT(
	Expected := expectedUnit,
	Actual := libResult.unit,
    Message := SEL(expectedUnit = libResult.unit,
	CONCAT('Pressure unit fail: exp = ',CONCAT( TO_STRING(expectedUnit), concat( ', act = ', TO_STRING(libResult.unit))))
    ,'test is ok')
);
END_METHOD

(*

short summary
==================
This test method tests ``ConvertPressure``
method of CNM_RecipeHandling library for special cases, 
it provides the possibility to handover test data via parameter 


.. <legal notes>

legal notes
=================
| SPDX-FileCopyrightText: © 2025 ekvip automation GmbH <info@ekvip.de>
| SPDX-License-Identifier: Apache-2.0
| For details check: Apache-2.0_

.. _Apache-2.0: https://www.apache.org/licenses/LICENSE-2.0

.. </legal notes>

parameters
==========

*)
METHOD testConvertPressureSpecialCases
VAR_INPUT
	(* The numeric pressure value to convert (e.g. 101325.0) *)
	sourceValue : LREAL;
	(* The original pressure unit (e.g. PASCAL, BAR) *)
	sourceUnit : CNM_RecipeHandling.PressureUnit;
	(*  Metric prefix for the input value (e.g. KILO, MILLI) *)
	sourcePrefix : CNM_RecipeHandling.MetricPrefixes;
	(* The expected result after conversion (e.g. 1.01325) *)
	expectedValue : LREAL;
	(* The target unit to which the pressure should be converted (e.g. BAR) *)
	expectedUnit :CNM_RecipeHandling.PressureUnit;
	(* Metric prefix for the expected result (e.g. NONE) *)
	expectedPrefix : CNM_RecipeHandling.MetricPrefixes;
END_VAR
VAR
	sourcePressure : CNM_RecipeHandling.Pressure;
	libResult : CNM_RecipeHandling.Pressure;
END_VAR
sourcePressure.value := sourceValue;
sourcePressure.unit := sourceUnit;
sourcePressure.prefix := sourcePrefix;

libResult := CNM_RecipeHandling.ConvertPressure(
	pressureToConvert :=sourcePressure,
	convertTo := expectedUnit,
	resultPrefix := expectedPrefix
);
IF Tc2_Utilities.LrealIsNaN(expectedValue) THEN
	AssertTrue(Condition := Tc2_Utilities.LrealIsNaN(libResult.value),
    Message := 'test faild assertion NaN should be true');
ELSIF NOT (Tc2_Utilities.LrealIsFinite(expectedValue))THEN
	 AssertTrue(Condition := NOT(Tc2_Utilities.LrealIsFinite(libResult.value)),
    Message := 'test faild assertion INF should be True');
END_IF
END_METHOD

(*

short summary
==================
This test method tests ``ConvertTemperature``
method of CNM_RecipeHandling library, 
it provides the possibility to handover test data via parameter 


.. <legal notes>

legal notes
=================
| SPDX-FileCopyrightText: © 2025 ekvip automation GmbH <info@ekvip.de>
| SPDX-License-Identifier: Apache-2.0
| For details check: Apache-2.0_

.. _Apache-2.0: https://www.apache.org/licenses/LICENSE-2.0

.. </legal notes>

parameters
==========

*)

METHOD testConvertTemprature
VAR_INPUT
	(* The numeric temperature value to be converted (e.g. 100.0) *)
	sourceValue : LREAL;
	(* The unit of the input temperature (e.g. DEGREE_CELSIUS, KELVIN) *)
	sourceUnit : CNM_RecipeHandling.TemperatureUnit;
	(* The expected result after conversion (e.g. 212.0) *)
	expectedValue : LREAL;
	(* The unit expected after conversion (e.g. DEGREE_FAHRENHEIT) *)
	expectedUnit :CNM_RecipeHandling.TemperatureUnit;
END_VAR
VAR
	sourceTemprature : CNM_RecipeHandling.Temperature;
	libResult : CNM_RecipeHandling.Temperature;
END_VAR
sourceTemprature.value := sourceValue;
sourceTemprature.unit := sourceUnit;

libResult := CNM_RecipeHandling.ConvertTemperature(
	temperatureToConvert := sourceTemprature,
	convertTo := expectedUnit,
);

THIS^.AssertEquals_LREAL(
    Expected := expectedValue,
    Actual := libResult.value,
    Delta := 0.01,
   Message := SEL(expectedValue = libResult.value,
	CONCAT('ConvertTemprature value fail: exp = ',CONCAT( TO_STRING(expectedValue), concat( ', act = ', TO_STRING(libResult.value))))
    ,'test is ok'));

THIS^.AssertEquals_INT(
	Expected := expectedUnit,
	Actual := libResult.unit,
    Message := SEL(expectedUnit = libResult.unit,
	CONCAT('ConvertTemprature unit fail: exp = ',CONCAT( TO_STRING(expectedUnit), concat( ', act = ', TO_STRING(libResult.unit))))
    ,'test is ok')
);
END_METHOD

(*

short summary
==================
This test method tests ``ConvertTemperature``
method of CNM_RecipeHandling library for special cases, 
it provides the possibility to handover test data via parameter 


.. <legal notes>

legal notes
=================
| SPDX-FileCopyrightText: © 2025 ekvip automation GmbH <info@ekvip.de>
| SPDX-License-Identifier: Apache-2.0
| For details check: Apache-2.0_

.. _Apache-2.0: https://www.apache.org/licenses/LICENSE-2.0

.. </legal notes>

parameters
==========

*)

METHOD testConvertTempratureSpecialCases
VAR_INPUT
	(* The numeric temperature value to be converted (e.g. 100.0) *)
	sourceValue : LREAL;
	(* The unit of the input temperature (e.g. DEGREE_CELSIUS, KELVIN) *)
	sourceUnit : CNM_RecipeHandling.TemperatureUnit;
	(* The expected result after conversion (e.g. 212.0) *)
	expectedValue : LREAL;
	(* The unit expected after conversion (e.g. DEGREE_FAHRENHEIT) *)
	expectedUnit :CNM_RecipeHandling.TemperatureUnit;
END_VAR
VAR
	sourceTemprature : CNM_RecipeHandling.Temperature;
	libResult : CNM_RecipeHandling.Temperature;
END_VAR
//test input
sourceTemprature.value := sourceValue;
sourceTemprature.unit := sourceUnit;

//function to call

libResult := CNM_RecipeHandling.ConvertTemperature(
	temperatureToConvert := sourceTemprature,
	convertTo := expectedUnit,
);
IF Tc2_Utilities.LrealIsNaN(expectedValue) THEN
	AssertTrue(Condition := Tc2_Utilities.LrealIsNaN(libResult.value),
    Message := 'test faild assertion NaN should be true');
ELSIF NOT (Tc2_Utilities.LrealIsFinite(expectedValue))THEN
	 AssertTrue(Condition := NOT(Tc2_Utilities.LrealIsFinite(libResult.value)),
    Message := 'test faild assertion INF should be True');
END_IF
END_METHOD

(*

short summary
==================
This test method tests ``ConvertVelocity``
method of CNM_RecipeHandling library, 
it provides the possibility to handover test data via parameter 


.. <legal notes>

legal notes
=================
| SPDX-FileCopyrightText: © 2025 ekvip automation GmbH <info@ekvip.de>
| SPDX-License-Identifier: Apache-2.0
| For details check: Apache-2.0_

.. _Apache-2.0: https://www.apache.org/licenses/LICENSE-2.0

.. </legal notes>

parameters
==========

*)

METHOD testConvertVelocity
VAR_INPUT
    (* Input velocity value to be converted, e.g. 10.0 *)
    sourceVelocityValue : LREAL; 

    (* Expected result after conversion, used for assertion *)
    expectedVelocityValue : LREAL;

    (* Unit of distance used in velocity, e.g. METER *)
    sourceUnit : CNM_RecipeHandling.LengthUnit;

    (* Metric prefix of the distance input, e.g. KILO *)
    sourceDistancePrefix : CNM_RecipeHandling.MetricPrefixes;

    (* Expected unit of distance after conversion *)
    expectedDistanceUnit : CNM_RecipeHandling.LengthUnit;

    (* Expected metric prefix for the converted distance *)
    expectedDistancePrefix : CNM_RecipeHandling.MetricPrefixes;

    (* Unit of time used in velocity, e.g. SECONDS *)
    sourceDurationUnit : CNM_RecipeHandling.DurationUnit;

    (* Metric prefix of the time input, e.g. MILLI *)
    sourceDurationPrefix : CNM_RecipeHandling.MetricPrefixes;

    (* Expected time unit after conversion *)
    expectedDurationUnit : CNM_RecipeHandling.DurationUnit;

    (* Expected time prefix after conversion *)
    expectedDurationPrefix : CNM_RecipeHandling.MetricPrefixes;

    (* Whether the assertion is expected to pass (TRUE) or fail (FALSE) *)
	assertionShouldBeTrue :BOOL;
END_VAR
VAR
	sourceDistance : CNM_RecipeHandling.Length;
	sourceDuration : CNM_RecipeHandling.Duration;
	sourceVelocity : CNM_RecipeHandling.Velocity;
	libResult : CNM_RecipeHandling.Velocity;
	sourcePrefix: CNM_RecipeHandling.MetricPrefixes;
END_VAR

//test-input
sourceVelocity.value := sourceVelocityValue;
sourceVelocity.distanceUnit := sourceUnit;
sourceVelocity.distancePrefix := sourceDistancePrefix;
sourceVelocity.timeUnit := sourceDurationUnit;
sourceVelocity.timePrefix := sourceDurationPrefix; 

sourceDistance.unit := sourceUnit;
sourceDistance.prefix := sourceDistancePrefix;
sourceDuration.unit := sourceDurationUnit;
sourceDuration.prefix := sourceDurationPrefix;

//function to call
libResult := CNM_RecipeHandling.ConvertVelocity(
	velocityToConvert:=sourceVelocity,
	convertDistanceTo :=expectedDistanceUnit,
	convertTimeTo := expectedDurationUnit,
	resultPrefixDistance := expectedDistancePrefix,
	resultPrefixTime := expectedDurationPrefix
);
THIS^.AssertEquals_LREAL(
    Expected := expectedVelocityValue,
    Actual := libResult.value,
    Delta := 0.01,
   Message := SEL(expectedVelocityValue = libResult.value,
	CONCAT('value fail: exp velocity value = ',CONCAT( TO_STRING(expectedVelocityValue), concat( ', act  velocity value = ', TO_STRING(libResult.value))))
    ,'test is ok'));


THIS^.AssertEquals_INT(
	Expected := expectedDistancePrefix,
	Actual := libResult.distancePrefix,
    Message := SEL(expectedDistancePrefix = libResult.distancePrefix,
	CONCAT('ConvertVelocity prefix fail: exp distance prefix  = ',CONCAT( TO_STRING(expectedDistancePrefix), concat( ', act distance prefix = ', TO_STRING(libResult.distancePrefix))))
    ,'test is ok')
);
THIS^.AssertEquals_INT(
	Expected := expectedDistanceUnit,
	Actual := libResult.distanceUnit,
    Message := SEL(expectedDistanceUnit = libResult.distanceUnit,
	CONCAT('ConvertVelocity unit fail: exp distance unit = ',CONCAT( TO_STRING(expectedDistanceUnit), concat( ', act distance unit = ', TO_STRING(libResult.distanceUnit))))
    ,'test is ok')
);

THIS^.AssertEquals_INT(
	Expected := expectedDurationPrefix,
	Actual := libResult.timePrefix,
    Message := SEL(expectedDurationPrefix = libResult.timePrefix,
	CONCAT('ConvertVelocity prefix fail: exp duration Prefix = ',CONCAT( TO_STRING(expectedDurationPrefix), concat( ', act duration Prefix = ', TO_STRING(libResult.timePrefix))))
    ,'test is ok')
);
THIS^.AssertEquals_INT(
	Expected := expectedDurationUnit,
	Actual := libResult.timeUnit,
    Message := SEL(expectedDurationUnit = libResult.timeUnit,
	CONCAT('ConvertVelocity unit fail: exp duration Unit = ',CONCAT( TO_STRING(expectedDurationUnit), concat( ', act duration Unit = ', TO_STRING(libResult.timeUnit))))
    ,'test is ok')
);
END_METHOD

(*

short summary
==================
This test method tests ``ConvertVelocity``
method of CNM_RecipeHandling library for special cases, 
it provides the possibility to handover test data via parameter 


.. <legal notes>

legal notes
=================
| SPDX-FileCopyrightText: © 2025 ekvip automation GmbH <info@ekvip.de>
| SPDX-License-Identifier: Apache-2.0
| For details check: Apache-2.0_

.. _Apache-2.0: https://www.apache.org/licenses/LICENSE-2.0

.. </legal notes>

parameters
==========

*)

METHOD testConvertVelocitySpecialCases
VAR_INPUT
    (* Input velocity value to be converted, e.g. 10.0 *)
    sourceVelocityValue : LREAL; 

    (* Expected result after conversion, used for assertion *)
    expectedVelocityValue : LREAL;

    (* Unit of distance used in velocity, e.g. METER *)
    sourceUnit : CNM_RecipeHandling.LengthUnit;

    (* Metric prefix of the distance input, e.g. KILO *)
    sourceDistancePrefix : CNM_RecipeHandling.MetricPrefixes;

    (* Expected unit of distance after conversion *)
    expectedDistanceUnit : CNM_RecipeHandling.LengthUnit;

    (* Expected metric prefix for the converted distance *)
    expectedDistancePrefix : CNM_RecipeHandling.MetricPrefixes;

    (* Unit of time used in velocity, e.g. SECONDS *)
    sourceDurationUnit : CNM_RecipeHandling.DurationUnit;

    (* Metric prefix of the time input, e.g. MILLI *)
    sourceDurationPrefix : CNM_RecipeHandling.MetricPrefixes;

    (* Expected time unit after conversion *)
    expectedDurationUnit : CNM_RecipeHandling.DurationUnit;

    (* Expected time prefix after conversion *)
    expectedDurationPrefix : CNM_RecipeHandling.MetricPrefixes;
END_VAR
VAR
	sourceDistance : CNM_RecipeHandling.Length;
	sourceDuration : CNM_RecipeHandling.Duration;
	sourceVelocity : CNM_RecipeHandling.Velocity;
	libResult : CNM_RecipeHandling.Velocity;
	sourcePrefix: CNM_RecipeHandling.MetricPrefixes;
END_VAR
//test-input
sourceVelocity.value := sourceVelocityValue;
sourceVelocity.distanceUnit := sourceUnit;
sourceVelocity.distancePrefix := sourceDistancePrefix;
sourceVelocity.timeUnit := sourceDurationUnit;
sourceVelocity.timePrefix := sourceDurationPrefix; 

sourceDistance.unit := sourceUnit;
sourceDistance.prefix := sourceDistancePrefix;
sourceDuration.unit := sourceDurationUnit;
sourceDuration.prefix := sourceDurationPrefix;

//function to call
libResult := CNM_RecipeHandling.ConvertVelocity(
	velocityToConvert:=sourceVelocity,
	convertDistanceTo :=expectedDistanceUnit,
	convertTimeTo := expectedDurationUnit,
	resultPrefixDistance := expectedDistancePrefix,
	resultPrefixTime := expectedDurationPrefix
);
IF Tc2_Utilities.LrealIsNaN(expectedVelocityValue) THEN
	AssertTrue(Condition := Tc2_Utilities.LrealIsNaN(libResult.value),
    Message := 'test faild assertion NaN should be true');
ELSIF NOT (Tc2_Utilities.LrealIsFinite(expectedVelocityValue))THEN
	 AssertTrue(Condition := NOT(Tc2_Utilities.LrealIsFinite(libResult.value)),
    Message := 'test faild assertion INF should be True');
END_IF
END_METHOD

(*

short summary
==================
This test method tests ``ConvertVolume``
method of CNM_RecipeHandling library, 
it provides the possibility to handover test data via parameter 


.. <legal notes>

legal notes
=================
| SPDX-FileCopyrightText: © 2025 ekvip automation GmbH <info@ekvip.de>
| SPDX-License-Identifier: Apache-2.0
| For details check: Apache-2.0_

.. _Apache-2.0: https://www.apache.org/licenses/LICENSE-2.0

.. </legal notes>

parameters
==========

*)

METHOD testConvertVolume
VAR_INPUT
    (* Input value to be converted, e.g. 1.0 *)
    sourceValue : LREAL;

    (* The unit of the input volume, e.g. LITER *)
    sourceUnit : CNM_RecipeHandling.VolumeUnit;

    (* Metric prefix for the input value, e.g. MILLI for milliliters *)
    sourcePrefix : CNM_RecipeHandling.MetricPrefixes;

    (* The expected result value after conversion *)
    expectedValue : LREAL;

    (* The expected unit after conversion, e.g. CUBIC_METER *)
    expectedUnit : CNM_RecipeHandling.VolumeUnit;

    (* The expected prefix for the converted result *)
    expectedPrefix : CNM_RecipeHandling.MetricPrefixes;
	
END_VAR
VAR
	sourceVolume : CNM_RecipeHandling.Volume;
	libResult : CNM_RecipeHandling.Volume;
END_VAR
sourceVolume.value := sourceValue;
sourceVolume.unit := sourceUnit;
sourceVolume.prefix := sourcePrefix;

libResult := CNM_RecipeHandling.ConvertVolume(
	volumeToConvert :=sourceVolume,
	convertTo := expectedUnit,
	resultPrefix := expectedPrefix
);

THIS^.AssertEquals_LREAL(
    Expected := expectedValue,
    Actual := libResult.value,
    Delta := 0.01,
   Message := SEL(expectedValue = libResult.value,
	CONCAT('Volume value fail: exp = ',CONCAT( TO_STRING(expectedValue), concat( ', act = ', TO_STRING(libResult.value))))
    ,'test is ok'));

THIS^.AssertEquals_INT(
	Expected := expectedPrefix,
	Actual := libResult.prefix,
    Message := SEL(expectedPrefix = libResult.prefix,
	CONCAT('Volume prefix fail: exp = ',CONCAT( TO_STRING(expectedPrefix), concat( ', act = ', TO_STRING(libResult.prefix))))
    ,'test is ok')
);

THIS^.AssertEquals_INT(
	Expected := expectedUnit,
	Actual := libResult.unit,
    Message := SEL(expectedUnit = libResult.unit,
	CONCAT('Volume unit fail: exp = ',CONCAT( TO_STRING(expectedUnit), concat( ', act = ', TO_STRING(libResult.unit))))
    ,'test is ok')
);
END_METHOD

(*

short summary
==================
This test method tests ``ConvertVolume``
method of CNM_RecipeHandling library for special cases, 
it provides the possibility to handover test data via parameter 


.. <legal notes>

legal notes
=================
| SPDX-FileCopyrightText: © 2025 ekvip automation GmbH <info@ekvip.de>
| SPDX-License-Identifier: Apache-2.0
| For details check: Apache-2.0_

.. _Apache-2.0: https://www.apache.org/licenses/LICENSE-2.0

.. </legal notes>

parameters
==========

*)

METHOD testConvertVolumeSpecialCases
VAR_INPUT
    (* Input value to be converted, e.g. 1.0 *)
    sourceValue : LREAL;

    (* The unit of the input volume, e.g. LITER *)
    sourceUnit : CNM_RecipeHandling.VolumeUnit;

    (* Metric prefix for the input value, e.g. MILLI for milliliters *)
    sourcePrefix : CNM_RecipeHandling.MetricPrefixes;

    (* The expected result value after conversion *)
    expectedValue : LREAL;

    (* The expected unit after conversion, e.g. CUBIC_METER *)
    expectedUnit : CNM_RecipeHandling.VolumeUnit;

    (* The expected prefix for the converted result *)
    expectedPrefix : CNM_RecipeHandling.MetricPrefixes;
END_VAR
VAR
	sourceVolume : CNM_RecipeHandling.Volume;
	libResult : CNM_RecipeHandling.Volume;
END_VAR
//teat-input
sourceVolume.value := sourceValue;
sourceVolume.unit := sourceUnit;
sourceVolume.prefix := sourcePrefix;

//function to call
libResult := CNM_RecipeHandling.ConvertVolume(
	volumeToConvert :=sourceVolume,
	convertTo := expectedUnit,
	resultPrefix := expectedPrefix
);
IF Tc2_Utilities.LrealIsNaN(expectedValue) THEN
	AssertTrue(Condition := Tc2_Utilities.LrealIsNaN(libResult.value),
    Message := 'test faild assertion NaN should be true');
ELSIF NOT (Tc2_Utilities.LrealIsFinite(expectedValue))THEN
	 AssertTrue(Condition := NOT(Tc2_Utilities.LrealIsFinite(libResult.value)),
    Message := 'test faild assertion INF should be True');
END_IF
END_METHOD

(*

short summary
==================
This test method tests ``ConvertWeight``
method of CNM_RecipeHandling library, 
it provides the possibility to handover test data via parameter 


.. <legal notes>

legal notes
=================
| SPDX-FileCopyrightText: © 2025 ekvip automation GmbH <info@ekvip.de>
| SPDX-License-Identifier: Apache-2.0
| For details check: Apache-2.0_

.. _Apache-2.0: https://www.apache.org/licenses/LICENSE-2.0

.. </legal notes>

parameters
==========

*)

METHOD testConvertWeight
VAR_INPUT
    (* The input weight value to convert, e.g. 1.0 *)
    sourceWeightValue : LREAL;

    (* The unit of the input weight, e.g. GRAM, KILOGRAM *)
    sourceWeightUnit : CNM_RecipeHandling.WeightUnit;

    (* Metric prefix for the input weight, e.g. MILLI, KILO *)
    sourcePrefix : CNM_RecipeHandling.MetricPrefixes;

    (* Expected result value after conversion *)
    expectedValue : LREAL;

    (* Expected unit of the converted weight *)
    expectedUnit : CNM_RecipeHandling.WeightUnit;

    (* Expected metric prefix of the result, e.g. NONE, KILO *)
    expectedPrefix : CNM_RecipeHandling.MetricPrefixes;
END_VAR
VAR
	sourceWeight : CNM_RecipeHandling.Weight;
	libResult : CNM_RecipeHandling.Weight;
END_VAR
sourceWeight.value := sourceWeightValue;
sourceWeight.unit := sourceWeightUnit;
sourceWeight.prefix := sourcePrefix;

libResult := CNM_RecipeHandling.ConvertWeight(
	weightToConvert := sourceWeight,
	convertTo := expectedUnit,
	resultPrefix := expectedPrefix
);

THIS^.AssertEquals_LREAL(
    Expected := expectedValue,
    Actual := libResult.value,
    Delta := 0.01,
   Message := SEL(expectedValue = libResult.value,
	CONCAT('value fail: exp Weight = ',CONCAT( TO_STRING(expectedValue), concat( ', act Weight = ', TO_STRING(libResult.value))))
    ,'test is ok'));

THIS^.AssertEquals_INT(
	Expected := expectedPrefix,
	Actual := libResult.prefix,
    Message := SEL(expectedPrefix = libResult.prefix,
	CONCAT('Weight prefix fail: exp = ',CONCAT( TO_STRING(expectedPrefix), concat( ', act = ', TO_STRING(libResult.prefix))))
    ,'test is ok')
);

THIS^.AssertEquals_INT(
	Expected := expectedUnit,
	Actual := libResult.unit,
    Message := SEL(expectedUnit = libResult.unit,
	CONCAT('Weight unit fail: exp = ',CONCAT( TO_STRING(expectedUnit), concat( ', act = ', TO_STRING(libResult.unit))))
    ,'Weight test is ok')
);
END_METHOD

(*

short summary
==================
This test method tests ``ConvertWeight``
method of CNM_RecipeHandling library for special cases, 
it provides the possibility to handover test data via parameter 


.. <legal notes>

legal notes
=================
| SPDX-FileCopyrightText: © 2025 ekvip automation GmbH <info@ekvip.de>
| SPDX-License-Identifier: Apache-2.0
| For details check: Apache-2.0_

.. _Apache-2.0: https://www.apache.org/licenses/LICENSE-2.0

.. </legal notes>

parameters
==========

*)

METHOD testConvertWightSpecialCases
VAR_INPUT
    (* The input weight value to convert, e.g. 1.0 *)
    sourceWeightValue : LREAL;

    (* The unit of the input weight, e.g. GRAM, KILOGRAM *)
    sourceWeightUnit : CNM_RecipeHandling.WeightUnit;

    (* Metric prefix for the input weight, e.g. MILLI, KILO *)
    sourcePrefix : CNM_RecipeHandling.MetricPrefixes;

    (* Expected result value after conversion *)
    expectedValue : LREAL;

    (* Expected unit of the converted weight *)
    expectedUnit : CNM_RecipeHandling.WeightUnit;

    (* Expected metric prefix of the result, e.g. NONE, KILO *)
    expectedPrefix : CNM_RecipeHandling.MetricPrefixes;
END_VAR
VAR
	sourceWeight : CNM_RecipeHandling.Weight;
	libResult : CNM_RecipeHandling.Weight;
END_VAR
sourceWeight.value := sourceWeightValue;
sourceWeight.unit := sourceWeightUnit;
sourceWeight.prefix := sourcePrefix;

libResult := CNM_RecipeHandling.ConvertWeight(
	weightToConvert := sourceWeight,
	convertTo := expectedUnit,
	resultPrefix := expectedPrefix
);

IF Tc2_Utilities.LrealIsNaN(expectedValue) THEN
	AssertTrue(Condition := Tc2_Utilities.LrealIsNaN(libResult.value),
    Message := 'test faild assertion NaN should be true');
ELSIF NOT (Tc2_Utilities.LrealIsFinite(expectedValue))THEN
	 AssertTrue(Condition := NOT(Tc2_Utilities.LrealIsFinite(libResult.value)),
    Message := 'test faild assertion INF should be True');
END_IF
END_METHOD

(*

short summary
==================
This test method tests ``CalculateVelocity``
method of CNM_RecipeHandling library, 
it provides the possibility to handover test data via parameter 


.. <legal notes>

legal notes
=================
| SPDX-FileCopyrightText: © 2025 ekvip automation GmbH <info@ekvip.de>
| SPDX-License-Identifier: Apache-2.0
| For details check: Apache-2.0_

.. _Apache-2.0: https://www.apache.org/licenses/LICENSE-2.0

.. </legal notes>

parameters
==========

*)

METHOD testFastPow10
VAR_INPUT
    (* The exponent to be tested, e.g. 3 for 10^3 *)
    exponentValue : INT;

    (* The expected result of 10 raised to the given exponent *)
    expectedFastPow10Value : LREAL;
END_VAR
VAR
	sourceExponenet : INT ;
	libResult : LREAL;
END_VAR
sourceExponenet := exponentValue;

libResult := CNM_RecipeHandling.FastPow10(
	exponent :=sourceExponenet,
);

THIS^.AssertEquals_LREAL(
    Expected := expectedFastPow10Value,
    Actual := libResult,
    Delta := 0.01,
   Message := SEL(expectedFastPow10Value = libResult,
	CONCAT('value fail: exp FastPow10 = ',CONCAT( TO_STRING(expectedFastPow10Value), concat( ', act FastPow10 value = ', TO_STRING(libResult))))
    ,'test is ok'));
END_METHOD

END_FUNCTION_BLOCK
